KUKA KRL program: ps_geo_c1.src, ps_geo_c1.dat

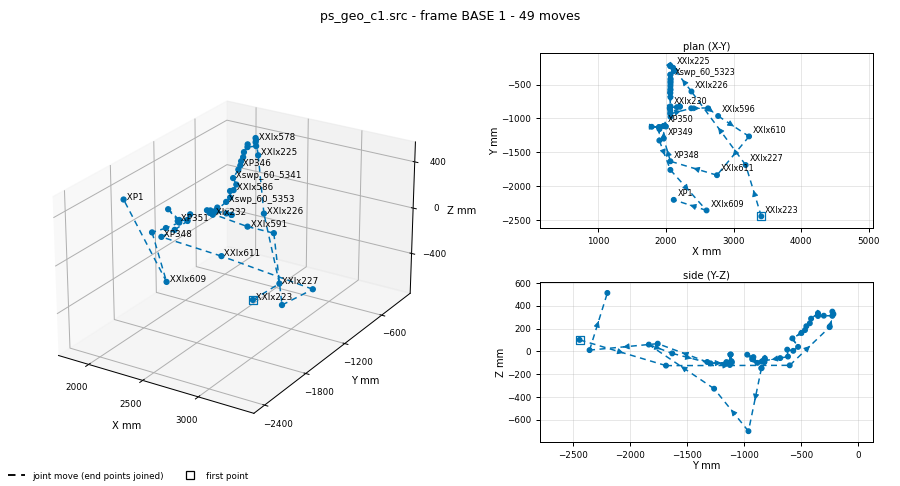
[picture p0: tool path of ps_geo_c1.src in frame BASE 1, 49 of 49 moves have a stored position in this frame; points joined in program order, loops and branches not executed]
--- ps_geo_c1.src ---
&ACCESS RVO1
&REL 105
&COMMENT Solda GUN C1 geometria
&PARAM DISKPATH = KRC:\R1\Program
DEF ps_geo_c1( )
;FOLD INI
  ;FOLD BASISTECH INI
    GLOBAL INTERRUPT DECL 3 WHEN $STOPMESS==TRUE DO IR_STOPM ( )
    INTERRUPT ON 3
    BAS (#INITMOV,0 )
  ;ENDFOLD (BASISTECH INI)
;FOLD SPOTTECH INI
USERSPOT(#INIT)
;ENDFOLD (SPOTTECH INI)
;FOLD GRIPPERTECH INI
USER_GRP(0,DUMMY,DUMMY,GDEFAULT)
;ENDFOLD (GRIPPERTECH INI)
  ;FOLD USER INI
    ;Make your modifications here

  ;ENDFOLD (USER INI)
;ENDFOLD (INI)

; Caracterização dos meios de produção:
; Versão Atual:
; 08/06/2013 12:00 Name: P13.050-R1 CHANGES: Solda Geometria Actros
; Gun C1 (F2 6640 0018 984)

chk_w2_wechs_ok ( )              ; CHECK C1

if MaxStandMenge (1) then
 MaxStandmengeErreicht (1)
endif

IF (NOT(GHOST())) THEN
if Elektrodenwechsel (1) then
 e_fraes2 ()
endif
ENDIF

;FOLD PTP Xlx223 CONT Vel=100 % P_OLP2 Tool[2]:GUN C1 Base[1]:Actros;%{PE}%R 8.2.20,%MKUKATPBASIS,%CMOVE,%VPTP,%P 1:PTP, 2:Xlx223, 3:C_DIS, 5:100, 7:P_OLP2
$BWDSTART=FALSE
PDAT_ACT=PP_OLP2
FDAT_ACT=FXlx223
BAS(#PTP_PARAMS,100)
PTP XXlx223 C_DIS
;ENDFOLD
;FOLD PTP Xlx227 CONT Vel=100 % P_OLP3 Tool[2]:GUN C1 Base[1]:Actros;%{PE}%R 8.2.20,%MKUKATPBASIS,%CMOVE,%VPTP,%P 1:PTP, 2:Xlx227, 3:C_DIS, 5:100, 7:P_OLP3
$BWDSTART=FALSE
PDAT_ACT=PP_OLP3
FDAT_ACT=FXlx227
BAS(#PTP_PARAMS,100)
PTP XXlx227 C_DIS
;ENDFOLD

;FOLD OUT 3339 'R1 solicita lib soldar geometria' State=TRUE ;%{PE}%R 8.2.20,%MKUKATPBASIS,%COUT,%VOUTX,%P 2:3339, 3:R1 solicita lib soldar geometria, 5:TRUE, 6:
$OUT[3339]=TRUE
;ENDFOLD
;FOLD WAIT FOR ( IN 3339 'Aguarda lib. Soldar geometria' );%{PE}%R 8.2.20,%MKUKATPBASIS,%CEXT_WAIT_FOR,%VEXT_WAIT_FOR,%P 2:, 4:, 5:$IN, 6:3339, 7:Aguarda lib. Soldar geometria, 9:
WAIT FOR  ( $IN[3339] )
;ENDFOLD
;FOLD OUT 3339 'R1 solicita lib soldar geometria' State=FALSE ;%{PE}%R 8.2.20,%MKUKATPBASIS,%COUT,%VOUTX,%P 2:3339, 3:R1 solicita lib soldar geometria, 5:FALSE, 6:
$OUT[3339]=FALSE
;ENDFOLD
;FOLD OUT 3348 'Fora area GEOBOX' State=FALSE ;%{PE}%R 8.2.20,%MKUKATPBASIS,%COUT,%VOUTX,%P 2:3348, 3:Fora area GEOBOX, 5:FALSE, 6:
$OUT[3348]=FALSE
;ENDFOLD

;FOLD PTP Xlx226 Vel=100 % P_OLP4 Tool[2]:GUN C1 Base[1]:Actros;%{PE}%R 8.2.20,%MKUKATPBASIS,%CMOVE,%VPTP,%P 1:PTP, 2:Xlx226, 3:, 5:100, 7:P_OLP4
$BWDSTART=FALSE
PDAT_ACT=PP_OLP4
FDAT_ACT=FXlx226
BAS(#PTP_PARAMS,100)
PTP XXlx226
;ENDFOLD

;FOLD Collision.Monitoring_AREA_6_On ;%{PE}%MKUKATPUSER
COLLSTOP( 12, 1 ) ;not Interrupt-Controlled
;ENDFOLD

;FOLD PTP Xlx225 CONT Vel=100 % P_OLP5 Tool[2]:GUN C1 Base[1]:Actros;%{PE}%R 8.2.20,%MKUKATPBASIS,%CMOVE,%VPTP,%P 1:PTP, 2:Xlx225, 3:C_DIS, 5:100, 7:P_OLP5
$BWDSTART=FALSE
PDAT_ACT=PP_OLP5
FDAT_ACT=FXlx225
BAS(#PTP_PARAMS,100)
PTP XXlx225 C_DIS
;ENDFOLD
;FOLD PTP Xlx578 CONT Vel=100 % PDAT1 Tool[2]:GUN C1 Base[1]:Actros;%{PE}%R 8.2.20,%MKUKATPBASIS,%CMOVE,%VPTP,%P 1:PTP, 2:Xlx578, 3:C_DIS, 5:100, 7:PDAT1
$BWDSTART=FALSE
PDAT_ACT=PPDAT1
FDAT_ACT=FXlx578
BAS(#PTP_PARAMS,100)
PTP XXlx578 C_DIS
;ENDFOLD

;FOLD ; swp_60_5311;%{PE}%R 8.2.20,%MKUKATPBASIS,%CCOMMENT,%VNORMAL,%P 2:swp_60_5311
;ENDFOLD
;FOLD PTP swp_60_5311 P_OLP6 SPOT Gun=1 RETR CLS PgNo1=26 ACTIVE=1 Tool[2]:GUN C1 Base[1]:Actros;%{PE}%R 8.2.2,%MKUKATPSPOT,%CSPOT,%VPTP,%P 1:PTP, 2:swp_60_5311, 3:, 5:100, 7:P_OLP6, 10:1, 12:#FIRST, 14:#CLO, 16:26, 18:1, 20:1, 22:0, 24:1, 25:S_OLP1
$BWDSTART=FALSE
PDAT_ACT=PP_OLP6
FDAT_ACT=Fswp_60_5311
BAS(#PTP_PARAMS,PP_OLP6.VEL)
S_ACT.GUN=1
S_ACT.PAIR=SDEFAULT.PAIR
S_ACT.RETR=#CLO
S_ACT.CLO_TM=1
S_ACT.PGNO1=26
S_ACT.PGNO2=SDEFAULT.PGNO2
S_ACT.PRESS1=SDEFAULT.PRESS1
S_ACT.PRESS2=SDEFAULT.PRESS2
S_READY=FALSE
PTP Xswp_60_5311
USERSPOT(#SPOT, S_ACT)
WAIT FOR S_READY
;ENDFOLD

;FOLD PTP Xlx583 CONT Vel=100 % PDAT6 Tool[2]:GUN C1 Base[1]:Actros;%{PE}%R 8.2.19,%MKUKATPBASIS,%CMOVE,%VPTP,%P 1:PTP, 2:Xlx583, 3:C_DIS, 5:100, 7:PDAT6
$BWDSTART=FALSE
PDAT_ACT=PPDAT6
FDAT_ACT=FXlx583
BAS(#PTP_PARAMS,100)
PTP XXlx583 C_DIS
;ENDFOLD
;FOLD PTP P347 CONT Vel=100 % PDAT39 Tool[2]:GUN C1 Base[1]:Actros;%{PE}%R 8.2.20,%MKUKATPBASIS,%CMOVE,%VPTP,%P 1:PTP, 2:P347, 3:C_DIS, 5:100, 7:PDAT39
$BWDSTART=FALSE
PDAT_ACT=PPDAT39
FDAT_ACT=FP347
BAS(#PTP_PARAMS,100)
PTP XP347 C_DIS
;ENDFOLD
;FOLD PTP Xlx584 CONT Vel=100 % PDAT7 Tool[2]:GUN C1 Base[1]:Actros;%{PE}%R 8.2.19,%MKUKATPBASIS,%CMOVE,%VPTP,%P 1:PTP, 2:Xlx584, 3:C_DIS, 5:100, 7:PDAT7
$BWDSTART=FALSE
PDAT_ACT=PPDAT7
FDAT_ACT=FXlx584
BAS(#PTP_PARAMS,100)
PTP XXlx584 C_DIS
;ENDFOLD

;FOLD ; swp_60_5317;%{PE}%R 8.2.20,%MKUKATPBASIS,%CCOMMENT,%VNORMAL,%P 2:swp_60_5317
;ENDFOLD
;FOLD PTP swp_60_5317 P_OLP42 SPOT Gun=1 RETR CLS PgNo1=27 ACTIVE=1 Tool[2]:GUN C1 Base[1]:Actros;%{PE}%R 8.2.2,%MKUKATPSPOT,%CSPOT,%VPTP,%P 1:PTP, 2:swp_60_5317, 3:, 5:100, 7:P_OLP42, 10:1, 12:#FIRST, 14:#CLO, 16:27, 18:1, 20:1, 22:0, 24:1, 25:S_OLP2
$BWDSTART=FALSE
PDAT_ACT=PP_OLP42
FDAT_ACT=Fswp_60_5317
BAS(#PTP_PARAMS,PP_OLP42.VEL)
S_ACT.GUN=1
S_ACT.PAIR=SDEFAULT.PAIR
S_ACT.RETR=#CLO
S_ACT.CLO_TM=1
S_ACT.PGNO1=27
S_ACT.PGNO2=SDEFAULT.PGNO2
S_ACT.PRESS1=SDEFAULT.PRESS1
S_ACT.PRESS2=SDEFAULT.PRESS2
S_READY=FALSE
PTP Xswp_60_5317
USERSPOT(#SPOT, S_ACT)
WAIT FOR S_READY
;ENDFOLD

;FOLD ; swp_60_5323;%{PE}%R 8.2.20,%MKUKATPBASIS,%CCOMMENT,%VNORMAL,%P 2:swp_60_5323
;ENDFOLD
;FOLD PTP swp_60_5323 P_OLP8 SPOT Gun=1 RETR CLS PgNo1=28 ACTIVE=1 Tool[2]:GUN C1 Base[1]:Actros;%{PE}%R 8.2.2,%MKUKATPSPOT,%CSPOT,%VPTP,%P 1:PTP, 2:swp_60_5323, 3:, 5:100, 7:P_OLP8, 10:1, 12:#FIRST, 14:#CLO, 16:28, 18:1, 20:1, 22:0, 24:1, 25:S_OLP3
$BWDSTART=FALSE
PDAT_ACT=PP_OLP8
FDAT_ACT=Fswp_60_5323
BAS(#PTP_PARAMS,PP_OLP8.VEL)
S_ACT.GUN=1
S_ACT.PAIR=SDEFAULT.PAIR
S_ACT.RETR=#CLO
S_ACT.CLO_TM=1
S_ACT.PGNO1=28
S_ACT.PGNO2=SDEFAULT.PGNO2
S_ACT.PRESS1=SDEFAULT.PRESS1
S_ACT.PRESS2=SDEFAULT.PRESS2
S_READY=FALSE
PTP Xswp_60_5323
USERSPOT(#SPOT, S_ACT)
WAIT FOR S_READY
;ENDFOLD

;FOLD PTP P345 CONT Vel=100 % PDAT37 Tool[2]:GUN C1 Base[1]:Actros;%{PE}%R 8.2.20,%MKUKATPBASIS,%CMOVE,%VPTP,%P 1:PTP, 2:P345, 3:C_DIS, 5:100, 7:PDAT37
$BWDSTART=FALSE
PDAT_ACT=PPDAT37
FDAT_ACT=FP345
BAS(#PTP_PARAMS,100)
PTP XP345 C_DIS
;ENDFOLD

;FOLD ; swp_60_5329;%{PE}%R 8.2.20,%MKUKATPBASIS,%CCOMMENT,%VNORMAL,%P 2:swp_60_5329
;ENDFOLD
;FOLD PTP swp_60_5329 P_OLP9 SPOT Gun=1 RETR CLS PgNo1=29 ACTIVE=1 Tool[2]:GUN C1 Base[1]:Actros;%{PE}%R 8.2.2,%MKUKATPSPOT,%CSPOT,%VPTP,%P 1:PTP, 2:swp_60_5329, 3:, 5:100, 7:P_OLP9, 10:1, 12:#FIRST, 14:#CLO, 16:29, 18:1, 20:1, 22:0, 24:1, 25:S_OLP4
$BWDSTART=FALSE
PDAT_ACT=PP_OLP9
FDAT_ACT=Fswp_60_5329
BAS(#PTP_PARAMS,PP_OLP9.VEL)
S_ACT.GUN=1
S_ACT.PAIR=SDEFAULT.PAIR
S_ACT.RETR=#CLO
S_ACT.CLO_TM=1
S_ACT.PGNO1=29
S_ACT.PGNO2=SDEFAULT.PGNO2
S_ACT.PRESS1=SDEFAULT.PRESS1
S_ACT.PRESS2=SDEFAULT.PRESS2
S_READY=FALSE
PTP Xswp_60_5329
USERSPOT(#SPOT, S_ACT)
WAIT FOR S_READY
;ENDFOLD

;FOLD PTP P346 CONT Vel=100 % PDAT38 Tool[2]:GUN C1 Base[1]:Actros;%{PE}%R 8.2.20,%MKUKATPBASIS,%CMOVE,%VPTP,%P 1:PTP, 2:P346, 3:C_DIS, 5:100, 7:PDAT38
$BWDSTART=FALSE
PDAT_ACT=PPDAT38
FDAT_ACT=FP346
BAS(#PTP_PARAMS,100)
PTP XP346 C_DIS
;ENDFOLD

;FOLD ; swp_60_5335;%{PE}%R 8.2.20,%MKUKATPBASIS,%CCOMMENT,%VNORMAL,%P 2:swp_60_5335
;ENDFOLD
;FOLD PTP swp_60_5335 P_OLP10 SPOT Gun=1 RETR CLS PgNo1=30 ACTIVE=1 Tool[2]:GUN C1 Base[1]:Actros;%{PE}%R 8.2.2,%MKUKATPSPOT,%CSPOT,%VPTP,%P 1:PTP, 2:swp_60_5335, 3:, 5:100, 7:P_OLP10, 10:1, 12:#FIRST, 14:#CLO, 16:30, 18:1, 20:1, 22:0, 24:1, 25:S_OLP5
$BWDSTART=FALSE
PDAT_ACT=PP_OLP10
FDAT_ACT=Fswp_60_5335
BAS(#PTP_PARAMS,PP_OLP10.VEL)
S_ACT.GUN=1
S_ACT.PAIR=SDEFAULT.PAIR
S_ACT.RETR=#CLO
S_ACT.CLO_TM=1
S_ACT.PGNO1=30
S_ACT.PGNO2=SDEFAULT.PGNO2
S_ACT.PRESS1=SDEFAULT.PRESS1
S_ACT.PRESS2=SDEFAULT.PRESS2
S_READY=FALSE
PTP Xswp_60_5335
USERSPOT(#SPOT, S_ACT)
WAIT FOR S_READY
;ENDFOLD

;FOLD ; swp_60_5341;%{PE}%R 8.2.20,%MKUKATPBASIS,%CCOMMENT,%VNORMAL,%P 2:swp_60_5341
;ENDFOLD
;FOLD PTP swp_60_5341 P_OLP11 SPOT Gun=1 RETR CLS PgNo1=31 ACTIVE=1 Tool[2]:GUN C1 Base[1]:Actros;%{PE}%R 8.2.2,%MKUKATPSPOT,%CSPOT,%VPTP,%P 1:PTP, 2:swp_60_5341, 3:, 5:100, 7:P_OLP11, 10:1, 12:#FIRST, 14:#CLO, 16:31, 18:1, 20:1, 22:0, 24:1, 25:S_OLP6
$BWDSTART=FALSE
PDAT_ACT=PP_OLP11
FDAT_ACT=Fswp_60_5341
BAS(#PTP_PARAMS,PP_OLP11.VEL)
S_ACT.GUN=1
S_ACT.PAIR=SDEFAULT.PAIR
S_ACT.RETR=#CLO
S_ACT.CLO_TM=1
S_ACT.PGNO1=31
S_ACT.PGNO2=SDEFAULT.PGNO2
S_ACT.PRESS1=SDEFAULT.PRESS1
S_ACT.PRESS2=SDEFAULT.PRESS2
S_READY=FALSE
PTP Xswp_60_5341
USERSPOT(#SPOT, S_ACT)
WAIT FOR S_READY
;ENDFOLD

;FOLD PTP Xlx585 CONT Vel=100 % PDAT8 Tool[2]:GUN C1 Base[1]:Actros;%{PE}%R 8.2.19,%MKUKATPBASIS,%CMOVE,%VPTP,%P 1:PTP, 2:Xlx585, 3:C_DIS, 5:100, 7:PDAT8
$BWDSTART=FALSE
PDAT_ACT=PPDAT8
FDAT_ACT=FXlx585
BAS(#PTP_PARAMS,100)
PTP XXlx585 C_DIS
;ENDFOLD
;FOLD PTP Xlx586 CONT Vel=100 % PDAT9 Tool[2]:GUN C1 Base[1]:Actros;%{PE}%R 8.2.19,%MKUKATPBASIS,%CMOVE,%VPTP,%P 1:PTP, 2:Xlx586, 3:C_DIS, 5:100, 7:PDAT9
$BWDSTART=FALSE
PDAT_ACT=PPDAT9
FDAT_ACT=FXlx586
BAS(#PTP_PARAMS,100)
PTP XXlx586 C_DIS
;ENDFOLD

;FOLD ; swp_60_5347;%{PE}%R 8.2.20,%MKUKATPBASIS,%CCOMMENT,%VNORMAL,%P 2:swp_60_5347
;ENDFOLD
;FOLD PTP swp_60_5347 P_OLP12 SPOT Gun=1 RETR CLS PgNo1=32 ACTIVE=1 Tool[2]:GUN C1 Base[1]:Actros;%{PE}%R 8.2.2,%MKUKATPSPOT,%CSPOT,%VPTP,%P 1:PTP, 2:swp_60_5347, 3:, 5:100, 7:P_OLP12, 10:1, 12:#FIRST, 14:#CLO, 16:32, 18:1, 20:1, 22:0, 24:1, 25:S_OLP7
$BWDSTART=FALSE
PDAT_ACT=PP_OLP12
FDAT_ACT=Fswp_60_5347
BAS(#PTP_PARAMS,PP_OLP12.VEL)
S_ACT.GUN=1
S_ACT.PAIR=SDEFAULT.PAIR
S_ACT.RETR=#CLO
S_ACT.CLO_TM=1
S_ACT.PGNO1=32
S_ACT.PGNO2=SDEFAULT.PGNO2
S_ACT.PRESS1=SDEFAULT.PRESS1
S_ACT.PRESS2=SDEFAULT.PRESS2
S_READY=FALSE
PTP Xswp_60_5347
USERSPOT(#SPOT, S_ACT)
WAIT FOR S_READY
;ENDFOLD

;FOLD PTP Xlx587 CONT Vel=100 % PDAT10 Tool[2]:GUN C1 Base[1]:Actros;%{PE}%R 8.2.19,%MKUKATPBASIS,%CMOVE,%VPTP,%P 1:PTP, 2:Xlx587, 3:C_DIS, 5:100, 7:PDAT10
$BWDSTART=FALSE
PDAT_ACT=PPDAT10
FDAT_ACT=FXlx587
BAS(#PTP_PARAMS,100)
PTP XXlx587 C_DIS
;ENDFOLD

;FOLD ; swp_60_5353;%{PE}%R 8.2.20,%MKUKATPBASIS,%CCOMMENT,%VNORMAL,%P 2:swp_60_5353
;ENDFOLD
;FOLD PTP swp_60_5353 P_OLP13 SPOT Gun=1 RETR CLS PgNo1=33 ACTIVE=1 Tool[2]:GUN C1 Base[1]:Actros;%{PE}%R 8.2.2,%MKUKATPSPOT,%CSPOT,%VPTP,%P 1:PTP, 2:swp_60_5353, 3:, 5:100, 7:P_OLP13, 10:1, 12:#FIRST, 14:#CLO, 16:33, 18:1, 20:1, 22:0, 24:1, 25:S_OLP8
$BWDSTART=FALSE
PDAT_ACT=PP_OLP13
FDAT_ACT=Fswp_60_5353
BAS(#PTP_PARAMS,PP_OLP13.VEL)
S_ACT.GUN=1
S_ACT.PAIR=SDEFAULT.PAIR
S_ACT.RETR=#CLO
S_ACT.CLO_TM=1
S_ACT.PGNO1=33
S_ACT.PGNO2=SDEFAULT.PGNO2
S_ACT.PRESS1=SDEFAULT.PRESS1
S_ACT.PRESS2=SDEFAULT.PRESS2
S_READY=FALSE
PTP Xswp_60_5353
USERSPOT(#SPOT, S_ACT)
WAIT FOR S_READY
;ENDFOLD

;FOLD PTP Xlx230 CONT Vel=100 % P_OLP14 Tool[2]:GUN C1 Base[1]:Actros;%{PE}%R 8.2.19,%MKUKATPBASIS,%CMOVE,%VPTP,%P 1:PTP, 2:Xlx230, 3:C_DIS, 5:100, 7:P_OLP14
$BWDSTART=FALSE
PDAT_ACT=PP_OLP14
FDAT_ACT=FXlx230
BAS(#PTP_PARAMS,100)
PTP XXlx230 C_DIS
;ENDFOLD

;FOLD PTP Xlx231 CONT Vel=100 % P_OLP43 Tool[2]:GUN C1 Base[1]:Actros;%{PE}%R 8.2.20,%MKUKATPBASIS,%CMOVE,%VPTP,%P 1:PTP, 2:Xlx231, 3:C_DIS, 5:100, 7:P_OLP43
$BWDSTART=FALSE
PDAT_ACT=PP_OLP43
FDAT_ACT=FXlx231
BAS(#PTP_PARAMS,100)
PTP XXlx231 C_DIS
;ENDFOLD
;FOLD PTP Xlx232 CONT Vel=100 % P_OLP44 Tool[2]:GUN C1 Base[1]:Actros;%{PE}%R 8.2.20,%MKUKATPBASIS,%CMOVE,%VPTP,%P 1:PTP, 2:Xlx232, 3:C_DIS, 5:100, 7:P_OLP44
$BWDSTART=FALSE
PDAT_ACT=PP_OLP44
FDAT_ACT=FXlx232
BAS(#PTP_PARAMS,100)
PTP XXlx232 C_DIS
;ENDFOLD
;FOLD Collision.Monitoring_AREA_6_Off . ;%{PE}%MKUKATPUSER
COLLSTOP( 12, 2+0 )
;ENDFOLD

;FOLD PTP Xlx229 CONT Vel=100 % P_OLP16 Tool[2]:GUN C1 Base[1]:Actros;%{PE}%R 8.2.19,%MKUKATPBASIS,%CMOVE,%VPTP,%P 1:PTP, 2:Xlx229, 3:C_DIS, 5:100, 7:P_OLP16
$BWDSTART=FALSE
PDAT_ACT=PP_OLP16
FDAT_ACT=FXlx229
BAS(#PTP_PARAMS,100)
PTP XXlx229 C_DIS
;ENDFOLD
;FOLD PTP Xlx228 CONT Vel=100 % P_OLP17 Tool[2]:GUN C1 Base[1]:Actros;%{PE}%R 8.2.19,%MKUKATPBASIS,%CMOVE,%VPTP,%P 1:PTP, 2:Xlx228, 3:C_DIS, 5:100, 7:P_OLP17
$BWDSTART=FALSE
PDAT_ACT=PP_OLP17
FDAT_ACT=FXlx228
BAS(#PTP_PARAMS,100)
PTP XXlx228 C_DIS
;ENDFOLD

;FOLD ; swp_60_5359;%{PE}%R 8.2.20,%MKUKATPBASIS,%CCOMMENT,%VNORMAL,%P 2:swp_60_5359
;ENDFOLD
;FOLD PTP swp_60_5359 P_OLP18 SPOT Gun=1 RETR CLS PgNo1=34 ACTIVE=1 Tool[2]:GUN C1 Base[1]:Actros;%{PE}%R 8.2.2,%MKUKATPSPOT,%CSPOT,%VPTP,%P 1:PTP, 2:swp_60_5359, 3:, 5:100, 7:P_OLP18, 10:1, 12:#FIRST, 14:#CLO, 16:34, 18:1, 20:1, 22:0, 24:1, 25:S_OLP9
$BWDSTART=FALSE
PDAT_ACT=PP_OLP18
FDAT_ACT=Fswp_60_5359
BAS(#PTP_PARAMS,PP_OLP18.VEL)
S_ACT.GUN=1
S_ACT.PAIR=SDEFAULT.PAIR
S_ACT.RETR=#CLO
S_ACT.CLO_TM=1
S_ACT.PGNO1=34
S_ACT.PGNO2=SDEFAULT.PGNO2
S_ACT.PRESS1=SDEFAULT.PRESS1
S_ACT.PRESS2=SDEFAULT.PRESS2
S_READY=FALSE
PTP Xswp_60_5359
USERSPOT(#SPOT, S_ACT)
WAIT FOR S_READY
;ENDFOLD

;FOLD PTP Xlx232 CONT Vel=100 % P_OLP19 Tool[2]:GUN C1 Base[1]:Actros;%{PE}%R8.2,%MKUKATPBASIS,%CMOVE,%VPTP,%P 1:PTP, 2:Xlx232, 3:C_DIS, 5:100, 7:P_OLP19
$BWDSTART = FALSE
PDAT_ACT= PP_OLP19
FDAT_ACT= Flx232
BAS(#PTP_PARAMS,100)
PTP Xlx232 C_DIS
;ENDFOLD
;FOLD PTP Xlx595 CONT Vel=100 % PDAT18 Tool[2]:GUN C1 Base[1]:Actros;%{PE}%R 8.2.19,%MKUKATPBASIS,%CMOVE,%VPTP,%P 1:PTP, 2:Xlx595, 3:C_DIS, 5:100, 7:PDAT18
$BWDSTART=FALSE
PDAT_ACT=PPDAT18
FDAT_ACT=FXlx595
BAS(#PTP_PARAMS,100)
PTP XXlx595 C_DIS
;ENDFOLD

;FOLD ; swp_60_5367;%{PE}%R 8.2.20,%MKUKATPBASIS,%CCOMMENT,%VNORMAL,%P 2:swp_60_5367
;ENDFOLD
;FOLD PTP swp_60_5367 P_OLP41 SPOT Gun=1 RETR CLS PgNo1=35 ACTIVE=1 Tool[2]:GUN C1 Base[1]:Actros;%{PE}%R 8.2.2,%MKUKATPSPOT,%CSPOT,%VPTP,%P 1:PTP, 2:swp_60_5367, 3:, 5:100, 7:P_OLP41, 10:1, 12:#FIRST, 14:#CLO, 16:35, 18:1, 20:1, 22:0, 24:1, 25:S_OLP14
$BWDSTART=FALSE
PDAT_ACT=PP_OLP41
FDAT_ACT=Fswp_60_5367
BAS(#PTP_PARAMS,PP_OLP41.VEL)
S_ACT.GUN=1
S_ACT.PAIR=SDEFAULT.PAIR
S_ACT.RETR=#CLO
S_ACT.CLO_TM=1
S_ACT.PGNO1=35
S_ACT.PGNO2=SDEFAULT.PGNO2
S_ACT.PRESS1=SDEFAULT.PRESS1
S_ACT.PRESS2=SDEFAULT.PRESS2
S_READY=FALSE
PTP Xswp_60_5367
USERSPOT(#SPOT, S_ACT)
WAIT FOR S_READY
;ENDFOLD

;FOLD PTP Xlx592 CONT Vel=100 % PDAT15 Tool[2]:GUN C1 Base[1]:Actros;%{PE}%R 8.2.19,%MKUKATPBASIS,%CMOVE,%VPTP,%P 1:PTP, 2:Xlx592, 3:C_DIS, 5:100, 7:PDAT15
$BWDSTART=FALSE
PDAT_ACT=PPDAT15
FDAT_ACT=FXlx592
BAS(#PTP_PARAMS,100)
PTP XXlx592 C_DIS
;ENDFOLD
;FOLD PTP Xlx591 CONT Vel=100 % PDAT14 Tool[2]:GUN C1 Base[1]:Actros;%{PE}%R 8.2.19,%MKUKATPBASIS,%CMOVE,%VPTP,%P 1:PTP, 2:Xlx591, 3:C_DIS, 5:100, 7:PDAT14
$BWDSTART=FALSE
PDAT_ACT=PPDAT14
FDAT_ACT=FXlx591
BAS(#PTP_PARAMS,100)
PTP XXlx591 C_DIS
;ENDFOLD
;FOLD PTP Xlx594 CONT Vel=100 % PDAT17 Tool[2]:GUN C1 Base[1]:Actros;%{PE}%R 8.2.19,%MKUKATPBASIS,%CMOVE,%VPTP,%P 1:PTP, 2:Xlx594, 3:C_DIS, 5:100, 7:PDAT17
$BWDSTART=FALSE
PDAT_ACT=PPDAT17
FDAT_ACT=FXlx594
BAS(#PTP_PARAMS,100)
PTP XXlx594 C_DIS
;ENDFOLD
;FOLD PTP Xlx596 CONT Vel=100 % PDAT19 Tool[2]:GUN C1 Base[1]:Actros;%{PE}%R 8.2.19,%MKUKATPBASIS,%CMOVE,%VPTP,%P 1:PTP, 2:Xlx596, 3:C_DIS, 5:100, 7:PDAT19
$BWDSTART=FALSE
PDAT_ACT=PPDAT19
FDAT_ACT=FXlx596
BAS(#PTP_PARAMS,100)
PTP XXlx596 C_DIS
;ENDFOLD
;FOLD PTP Xlx610 CONT Vel=100 % PDAT33 Tool[2]:GUN C1 Base[1]:Actros;%{PE}%R 8.2.19,%MKUKATPBASIS,%CMOVE,%VPTP,%P 1:PTP, 2:Xlx610, 3:C_DIS, 5:100, 7:PDAT33
$BWDSTART=FALSE
PDAT_ACT=PPDAT33
FDAT_ACT=FXlx610
BAS(#PTP_PARAMS,100)
PTP XXlx610 C_DIS
;ENDFOLD
;FOLD PTP Xlx611 CONT Vel=100 % PDAT34 Tool[2]:GUN C1 Base[1]:Actros;%{PE}%R 8.2.19,%MKUKATPBASIS,%CMOVE,%VPTP,%P 1:PTP, 2:Xlx611, 3:C_DIS, 5:100, 7:PDAT34
$BWDSTART=FALSE
PDAT_ACT=PPDAT34
FDAT_ACT=FXlx611
BAS(#PTP_PARAMS,100)
PTP XXlx611 C_DIS
;ENDFOLD
;FOLD PTP P348 CONT Vel=100 % PDAT40 Tool[2]:GUN C1 Base[1]:Actros;%{PE}%R 8.2.20,%MKUKATPBASIS,%CMOVE,%VPTP,%P 1:PTP, 2:P348, 3:C_DIS, 5:100, 7:PDAT40
$BWDSTART=FALSE
PDAT_ACT=PPDAT40
FDAT_ACT=FP348
BAS(#PTP_PARAMS,100)
PTP XP348 C_DIS
;ENDFOLD
;FOLD PTP P349 CONT Vel=100 % PDAT41 Tool[2]:GUN C1 Base[1]:Actros;%{PE}%R 8.2.20,%MKUKATPBASIS,%CMOVE,%VPTP,%P 1:PTP, 2:P349, 3:C_DIS, 5:100, 7:PDAT41
$BWDSTART=FALSE
PDAT_ACT=PPDAT41
FDAT_ACT=FP349
BAS(#PTP_PARAMS,100)
PTP XP349 C_DIS
;ENDFOLD
;FOLD PTP P350 PDAT42 RETR CLS Gun=1 Tool[2]:GUN C1 Base[1]:Actros;%{PE}%R 8.2.2,%MKUKATPSPOT,%CRETR,%VPTP,%P 1:PTP, 2:P350, 3:, 5:100, 7:PDAT42, 9:#CLO, 11:1, 13:#FIRST
$BWDSTART=FALSE
PDAT_ACT=PPDAT42
FDAT_ACT=FP350
BAS(#PTP_PARAMS,PPDAT42.VEL)
S_ACT.GUN=1
S_ACT.PAIR=#FIRST
S_ACT.RETR=#CLO
S_READY=FALSE
PTP XP350
USERSPOT(#RETR, S_ACT)
WAIT FOR S_READY
;ENDFOLD

;FOLD ; swp_60_5377;%{PE}%R 8.2.20,%MKUKATPBASIS,%CCOMMENT,%VNORMAL,%P 2:swp_60_5377
;ENDFOLD
;FOLD PTP SWP_60_5377 PDAT43 SPOT Gun=1 RETR CLS PgNo1=36 ACTIVE=1 Tool[2]:GUN C1 Base[1]:Actros;%{PE}%R 8.2.2,%MKUKATPSPOT,%CSPOT,%VPTP,%P 1:PTP, 2:SWP_60_5377, 3:, 5:100, 7:PDAT43, 10:1, 12:#FIRST, 14:#CLO, 16:36, 18:1, 20:0, 22:0, 24:1, 25:SDAT1
$BWDSTART=FALSE
PDAT_ACT=PPDAT43
FDAT_ACT=FSWP_60_5377
BAS(#PTP_PARAMS,PPDAT43.VEL)
S_ACT.GUN=1
S_ACT.PAIR=SDEFAULT.PAIR
S_ACT.RETR=#CLO
S_ACT.CLO_TM=1
S_ACT.PGNO1=36
S_ACT.PGNO2=SDEFAULT.PGNO2
S_ACT.PRESS1=SDEFAULT.PRESS1
S_ACT.PRESS2=SDEFAULT.PRESS2
S_READY=FALSE
PTP XSWP_60_5377
USERSPOT(#SPOT, S_ACT)
WAIT FOR S_READY
;ENDFOLD

;FOLD PTP P456 CONT Vel=100 % PDAT44 Tool[2]:GUN C1 Base[1]:Actros;%{PE}%R 8.2.20,%MKUKATPBASIS,%CMOVE,%VPTP,%P 1:PTP, 2:P456, 3:C_DIS, 5:100, 7:PDAT44
$BWDSTART=FALSE
PDAT_ACT=PPDAT44
FDAT_ACT=FP456
BAS(#PTP_PARAMS,100)
PTP XP456 C_DIS
;ENDFOLD
;FOLD PTP P351 CONT Vel=100 % PDAT45 Tool[2]:GUN C1 Base[1]:Actros;%{PE}%R 8.2.20,%MKUKATPBASIS,%CMOVE,%VPTP,%P 1:PTP, 2:P351, 3:C_DIS, 5:100, 7:PDAT45
$BWDSTART=FALSE
PDAT_ACT=PPDAT45
FDAT_ACT=FP351
BAS(#PTP_PARAMS,100)
PTP XP351 C_DIS
;ENDFOLD
;FOLD PTP P352 CONT Vel=100 % PDAT46 Tool[2]:GUN C1 Base[1]:Actros;%{PE}%R 8.2.20,%MKUKATPBASIS,%CMOVE,%VPTP,%P 1:PTP, 2:P352, 3:C_DIS, 5:100, 7:PDAT46
$BWDSTART=FALSE
PDAT_ACT=PPDAT46
FDAT_ACT=FP352
BAS(#PTP_PARAMS,100)
PTP XP352 C_DIS
;ENDFOLD

;FOLD ; swp_60_5387;%{PE}%R 8.2.20,%MKUKATPBASIS,%CCOMMENT,%VNORMAL,%P 2:swp_60_5387
;ENDFOLD
;FOLD PTP SWP_60_5387 PDAT47 SPOT Gun=1 RETR CLS PgNo1=37 ACTIVE=1 Tool[2]:GUN C1 Base[1]:Actros;%{PE}%R 8.2.2,%MKUKATPSPOT,%CSPOT,%VPTP,%P 1:PTP, 2:SWP_60_5387, 3:, 5:100, 7:PDAT47, 10:1, 12:#FIRST, 14:#CLO, 16:37, 18:1, 20:0, 22:0, 24:1, 25:SDAT2
$BWDSTART=FALSE
PDAT_ACT=PPDAT47
FDAT_ACT=FSWP_60_5387
BAS(#PTP_PARAMS,PPDAT47.VEL)
S_ACT.GUN=1
S_ACT.PAIR=SDEFAULT.PAIR
S_ACT.RETR=#CLO
S_ACT.CLO_TM=1
S_ACT.PGNO1=37
S_ACT.PGNO2=SDEFAULT.PGNO2
S_ACT.PRESS1=SDEFAULT.PRESS1
S_ACT.PRESS2=SDEFAULT.PRESS2
S_READY=FALSE
PTP XSWP_60_5387
USERSPOT(#SPOT, S_ACT)
WAIT FOR S_READY
;ENDFOLD

;FOLD PTP P455 CONT Vel=100 % PDAT48 Tool[2]:GUN C1 Base[1]:Actros;%{PE}%R 8.2.20,%MKUKATPBASIS,%CMOVE,%VPTP,%P 1:PTP, 2:P455, 3:C_DIS, 5:100, 7:PDAT48
$BWDSTART=FALSE
PDAT_ACT=PPDAT48
FDAT_ACT=FP455
BAS(#PTP_PARAMS,100)
PTP XP455 C_DIS
;ENDFOLD
;FOLD PTP P457 CONT Vel=100 % PDAT49 Tool[2]:GUN C1 Base[1]:Actros;%{PE}%R 8.2.20,%MKUKATPBASIS,%CMOVE,%VPTP,%P 1:PTP, 2:P457, 3:C_DIS, 5:100, 7:PDAT49
$BWDSTART=FALSE
PDAT_ACT=PPDAT49
FDAT_ACT=FP457
BAS(#PTP_PARAMS,100)
PTP XP457 C_DIS
;ENDFOLD
;FOLD PTP P458 CONT Vel=100 % PDAT50 Tool[2]:GUN C1 Base[1]:Actros;%{PE}%R 8.2.20,%MKUKATPBASIS,%CMOVE,%VPTP,%P 1:PTP, 2:P458, 3:C_DIS, 5:100, 7:PDAT50
$BWDSTART=FALSE
PDAT_ACT=PPDAT50
FDAT_ACT=FP458
BAS(#PTP_PARAMS,100)
PTP XP458 C_DIS
;ENDFOLD
;FOLD PTP Xlx609 CONT Vel=100 % PDAT32 Tool[2]:GUN C1 Base[1]:Actros;%{PE}%R 8.2.20,%MKUKATPBASIS,%CMOVE,%VPTP,%P 1:PTP, 2:Xlx609, 3:C_DIS, 5:100, 7:PDAT32
$BWDSTART=FALSE
PDAT_ACT=PPDAT32
FDAT_ACT=FXlx609
BAS(#PTP_PARAMS,100)
PTP XXlx609 C_DIS
;ENDFOLD
;FOLD PTP P1 Vel=100 % PDAT53 Tool[2]:GUN C1 Base[1]:Actros;%{PE}%R 8.2.20,%MKUKATPBASIS,%CMOVE,%VPTP,%P 1:PTP, 2:P1, 3:, 5:100, 7:PDAT53
$BWDSTART=FALSE
PDAT_ACT=PPDAT53
FDAT_ACT=FP1
BAS(#PTP_PARAMS,100)
PTP XP1
;ENDFOLD

;FOLD OUT 3348 'Fora area GEOBOX' State=TRUE ;%{PE}%R 8.2.20,%MKUKATPBASIS,%COUT,%VOUTX,%P 2:3348, 3:Fora area GEOBOX, 5:TRUE, 6:
$OUT[3348]=TRUE
;ENDFOLD

IF (NOT(GHOST())) THEN
if FraesAnf (1) then
 f_fraes2 ()
endif
ENDIF
END

--- ps_geo_c1.dat ---
&ACCESS RVO1
&REL 105
&COMMENT Solda GUN C1 geometria
&PARAM DISKPATH = KRC:\R1\Program
DEFDAT  ps_geo_c1
;FOLD EXTERNAL DECLARATIONS;%{PE}%MKUKATPBASIS,%CEXT,%VCOMMON,%P
;FOLD GRIPPERTECH EXT
EXT  H50 (INT  :IN,INT  :IN,INT  :IN,GRP_TYP  :IN )
;ENDFOLD (GRIPPERTECH EXT)
;FOLD SPOTTECH EXT
EXT  USERSPOT (S_COMMAND  :IN,SPOT_TYPE  :IN )
;ENDFOLD (SPOTTECH EXT)
;FOLD BASISTECH EXT;%{PE}%MKUKATPBASIS,%CEXT,%VEXT,%P
EXT  BAS (BAS_COMMAND  :IN,REAL  :IN )
DECL INT SUCCESS
;ENDFOLD (BASISTECH EXT)
;FOLD USER EXT;%{E}%MKUKATPUSER,%CEXT,%VEXT,%P
;Make your modifications here

;ENDFOLD (USER EXT)
;ENDFOLD (EXTERNAL DECLARATIONS)

;# ============ START PATH : swp_p13050r1_l_geo_c1 =============
DECL PDAT PP_OLP2={VEL 100.0,ACC 100.0,APO_DIST 100.0,APO_MODE #CDIS}
DECL PDAT PP_OLP3={VEL 100.0,ACC 100.0,APO_DIST 100.0,APO_MODE #CDIS}
DECL PDAT PP_OLP4={VEL 100.0,ACC 100.0,APO_DIST 100.0,APO_MODE #CDIS}
DECL PDAT PP_OLP5={VEL 100.0,ACC 100.0,APO_DIST 100.0,APO_MODE #CDIS}
DECL FDAT Fswp_60_5311={TOOL_NO 2,BASE_NO 1,IPO_FRAME #BASE,POINT2[] " ",TQ_STATE FALSE}
DECL PDAT PP_OLP6={VEL 100.0,ACC 100.0,APO_DIST 0.0}
DECL SPOT_TYPE SS_OLP1={GUN 1,PAIR #FIRST,RETR #CLO,CLO_TM 0,PGNO1 1,PRESS1 1.0,PGNO2 0,PRESS2 0.0}
DECL E6POS Xswp_60_5311={X 2065.98511,Y -226.899902,Z 349.511993,A 110.327499,B -85.6865234,C 69.4538727,S 2,T 42,E1 -4474.354,E2 0.0,E3 0.0,E4 0.0,E5 0.0,E6 0.0}
DECL FDAT Fswp_60_5317={TOOL_NO 2,BASE_NO 1,IPO_FRAME #BASE,POINT2[] " ",TQ_STATE FALSE}
DECL SPOT_TYPE SS_OLP2={GUN 1,PAIR #FIRST,RETR #CLO,CLO_TM 0,PGNO1 1,PRESS1 1.0,PGNO2 0,PRESS2 0.0}
DECL E6POS Xswp_60_5317={X 2067.58789,Y -353.265594,Z 335.725708,A -98.2681732,B -88.2489166,C -79.6126328,S 2,T 42,E1 -4219.60889,E2 0.0,E3 0.0,E4 0.0,E5 0.0,E6 0.0}
DECL FDAT Fswp_60_5323={TOOL_NO 2,BASE_NO 1,IPO_FRAME #BASE,POINT2[] " ",TQ_STATE FALSE}
DECL PDAT PP_OLP8={VEL 100.0,ACC 100.0,APO_DIST 0.0}
DECL SPOT_TYPE SS_OLP3={GUN 1,PAIR #FIRST,RETR #CLO,CLO_TM 0,PGNO1 1,PRESS1 1.0,PGNO2 0,PRESS2 0.0}
DECL E6POS Xswp_60_5323={X 2069.21704,Y -413.284393,Z 287.633209,A -84.5369034,B -66.7329865,C -93.644577,S 2,T 42,E1 -4219.93799,E2 0.0,E3 0.0,E4 0.0,E5 0.0,E6 0.0}
DECL FDAT Fswp_60_5329={TOOL_NO 2,BASE_NO 1,IPO_FRAME #BASE,POINT2[] " ",TQ_STATE FALSE}
DECL PDAT PP_OLP9={VEL 100.0,ACC 100.0,APO_DIST 0.0}
DECL SPOT_TYPE SS_OLP4={GUN 1,PAIR #FIRST,RETR #CLO,CLO_TM 0,PGNO1 1,PRESS1 1.0,PGNO2 0,PRESS2 0.0}
DECL E6POS Xswp_60_5329={X 2068.11792,Y -455.172089,Z 221.144104,A -83.784668,B -70.5104675,C -94.3365021,S 2,T 42,E1 -4219.93799,E2 0.0,E3 0.0,E4 0.0,E5 0.0,E6 0.0}
DECL FDAT Fswp_60_5335={TOOL_NO 2,BASE_NO 1,IPO_FRAME #BASE,POINT2[] " ",TQ_STATE FALSE}
DECL PDAT PP_OLP10={VEL 100.0,ACC 100.0,APO_DIST 0.0}
DECL SPOT_TYPE SS_OLP5={GUN 1,PAIR #FIRST,RETR #CLO,CLO_TM 0,PGNO1 1,PRESS1 1.0,PGNO2 0,PRESS2 0.0}
DECL E6POS Xswp_60_5335={X 2068.32104,Y -498.486511,Z 162.031601,A -83.1203003,B -73.1582031,C -94.9776001,S 2,T 42,E1 -4219.93799,E2 0.0,E3 0.0,E4 0.0,E5 0.0,E6 0.0}
DECL FDAT Fswp_60_5341={TOOL_NO 2,BASE_NO 1,IPO_FRAME #BASE,POINT2[] " "}
DECL PDAT PP_OLP11={VEL 100.0,ACC 100.0,APO_DIST 0.0}
DECL SPOT_TYPE SS_OLP6={GUN 1,PAIR #FIRST,RETR #CLO,CLO_TM 0,PGNO1 1,PRESS1 1.0,PGNO2 0,PRESS2 0.0}
DECL E6POS Xswp_60_5341={X 2067.21704,Y -577.190186,Z 114.618599,A -85.77388,B -55.6890182,C -92.5561829,S 2,T 10,E1 -4219.93799,E2 0.0,E3 0.0,E4 0.0,E5 0.0,E6 0.0}
DECL FDAT Fswp_60_5347={TOOL_NO 2,BASE_NO 1,IPO_FRAME #BASE,POINT2[] " ",TQ_STATE FALSE}
DECL PDAT PP_OLP12={VEL 100.0,ACC 100.0,APO_DIST 0.0}
DECL SPOT_TYPE SS_OLP7={GUN 1,PAIR #FIRST,RETR #CLO,CLO_TM 0,PGNO1 1,PRESS1 1.0,PGNO2 0,PRESS2 0.0}
DECL E6POS Xswp_60_5347={X 2066.55298,Y -622.881287,Z 15.8281803,A -85.6193771,B -57.4586182,C -92.6872101,S 2,T 10,E1 -4219.9458,E2 0.0,E3 0.0,E4 0.0,E5 0.0,E6 0.0}
DECL FDAT Fswp_60_5353={TOOL_NO 2,BASE_NO 1,IPO_FRAME #BASE,POINT2[] " "}
DECL PDAT PP_OLP13={VEL 100.0,ACC 100.0,APO_DIST 0.0}
DECL SPOT_TYPE SS_OLP8={GUN 1,PAIR #FIRST,RETR #CLO,CLO_TM 0,PGNO1 1,PRESS1 1.0,PGNO2 0,PRESS2 0.0}
DECL E6POS Xswp_60_5353={X 2067.23193,Y -684.528625,Z -58.5064888,A -86.9186478,B -33.8480606,C -91.7377472,S 2,T 10,E1 -4219.99512,E2 0.0,E3 0.0,E4 0.0,E5 0.0,E6 0.0}
DECL PDAT PP_OLP14={VEL 100.0,ACC 100.0,APO_DIST 100.0,APO_MODE #CDIS}
DECL PDAT PP_OLP16={VEL 100.0,ACC 100.0,APO_DIST 100.0,APO_MODE #CDIS}
DECL PDAT PP_OLP17={VEL 100.0,ACC 100.0,APO_DIST 100.0,APO_MODE #CDIS}
DECL FDAT Fswp_60_5359={TOOL_NO 2,BASE_NO 1,IPO_FRAME #BASE,POINT2[] " ",TQ_STATE FALSE}
DECL PDAT PP_OLP18={VEL 100.0,ACC 100.0,APO_DIST 0.0}
DECL SPOT_TYPE SS_OLP9={GUN 1,PAIR #FIRST,RETR #CLO,CLO_TM 0,PGNO1 1,PRESS1 1.0,PGNO2 0,PRESS2 0.0}
DECL E6POS Xswp_60_5359={X 2067.65308,Y -819.673706,Z -59.9566994,A 89.9988708,B -35.2867393,C 90.0017166,S 2,T 42,E1 -4487.30518,E2 0.0,E3 0.0,E4 0.0,E5 0.0,E6 0.0}
DECL FDAT Flx232={TOOL_NO 2,BASE_NO 1,IPO_FRAME #BASE,POINT2[] " "}
DECL PDAT PP_OLP19={VEL 100.0,ACC 100.0,APO_DIST 100.0,APO_MODE #CDIS}
DECL E6POS Xlx232={X 2065.2561,Y -885.252014,Z -100.142998,A 90.0,B -35.6880989,C 90.0,S 2,T 42,E1 -4487.2998,E2 0.0,E3 0.0,E4 0.0,E5 0.0,E6 0.0}
DECL FDAT Fswp_60_5367={TOOL_NO 2,BASE_NO 1,IPO_FRAME #BASE,POINT2[] " "}
DECL SPOT_TYPE SS_OLP10={GUN 1,PAIR #FIRST,RETR #CLO,CLO_TM 0,PGNO1 1,PRESS1 1.0,PGNO2 0,PRESS2 0.0}
DECL E6POS Xswp_60_5367={X 2067.479,Y -973.934082,Z -28.4924908,A 89.9911804,B -81.1077728,C 90.0090179,S 2,T 42,E1 -4487.2998,E2 0.0,E3 0.0,E4 0.0,E5 0.0,E6 0.0}
DECL FDAT Fswp_60_5377={TOOL_NO 2,BASE_NO 1,IPO_FRAME #BASE,POINT2[] " "}
DECL SPOT_TYPE SS_OLP11={GUN 1,PAIR #FIRST,RETR #CLO,CLO_TM 0,PGNO1 1,PRESS1 1.0,PGNO2 0,PRESS2 0.0}
DECL E6POS Xswp_60_5377={X 2000.44202,Y -1118.71997,Z -26.2877502,A -0.164200798,B -46.8474388,C 88.6065521,S 2,T 2,E1 -3882.23608,E2 0.0,E3 0.0,E4 0.0,E5 0.0,E6 0.0}
DECL SPOT_TYPE SS_OLP12={GUN 1,PAIR #FIRST,RETR #CLO,CLO_TM 0,PGNO1 1,PRESS1 1.0,PGNO2 0,PRESS2 0.0}
DECL BASIS_SUGG_T LAST_BASIS={POINT1[] "P0                      ",POINT2[] "P0                      ",CP_PARAMS[] "CPDAT0                  ",PTP_PARAMS[] "PDAT0                   ",CONT[] "                        ",CP_VEL[] "2.0                     ",PTP_VEL[] " 100                    ",SYNC_PARAMS[] "SYNCDAT                 ",SPL_NAME[] "S0                      "}
DECL E6POS XXLX223={X 3409.55396,Y -2445.41089,Z 101.454399,A 10.5907497,B 25.0754108,C 8.57579041,S 2,T 2,E1 -2854.21997,E2 0.0,E3 0.0,E4 0.0,E5 0.0,E6 0.0}
DECL FDAT FXlx223={TOOL_NO 2,BASE_NO 1,IPO_FRAME #BASE,POINT2[] " ",TQ_STATE FALSE}
DECL E6POS XXLX227={X 3178.82104,Y -1687.01099,Z -124.4701,A -38.8299904,B 13.9388504,C -8.95322132,S 2,T 10,E1 -4153.19482,E2 0.0,E3 0.0,E4 0.0,E5 0.0,E6 0.0}
DECL FDAT FXlx227={TOOL_NO 2,BASE_NO 1,IPO_FRAME #BASE,POINT2[] " ",TQ_STATE FALSE}
DECL E6POS XXLX226={X 2377.62109,Y -600.91333,Z -122.117203,A -174.316498,B -60.562809,C -1.327986,S 2,T 42,E1 -4433.27295,E2 0.0,E3 0.0,E4 0.0,E5 0.0,E6 0.0}
DECL FDAT FXlx226={TOOL_NO 2,BASE_NO 1,IPO_FRAME #BASE,POINT2[] " ",TQ_STATE FALSE}
DECL E6POS XXLX225={X 2106.66602,Y -251.165894,Z 213.202896,A 110.725197,B -85.6747131,C 65.7768402,S 2,T 42,E1 -4474.38721,E2 0.0,E3 0.0,E4 0.0,E5 0.0,E6 0.0}
DECL FDAT FXlx225={TOOL_NO 2,BASE_NO 1,IPO_FRAME #BASE,POINT2[] " ",TQ_STATE FALSE}
DECL E6POS XXLX578={X 2064.31494,Y -217.566193,Z 327.9534,A 110.3564,B -85.6859436,C 69.4285126,S 2,T 42,E1 -4474.38477,E2 0.0,E3 0.0,E4 0.0,E5 0.0,E6 0.0}
DECL FDAT FXlx578={TOOL_NO 2,BASE_NO 1,IPO_FRAME #BASE,POINT2[] " ",TQ_STATE FALSE}
DECL PDAT PPDAT1={VEL 100.0,ACC 100.0,APO_DIST 100.0,APO_MODE #CDIS}
DECL SPOT_SUGG_T LAST_SPOT={GUN[] "1                       ",RETR_CMD[] "#CLO                    ",CHOISE[] "#FIRST                  ",CLO_TM[] "1                       ",PGNO1[] "1                       ",PRESS1[] "0                       ",PGNO2[] "1                       ",PRESS2[] "0                       ",SPOT_PARAMS[] "SDAT2                   "}
DECL PDAT PPDAT6={VEL 100.0,ACC 100.0,APO_DIST 100.0,APO_MODE #CDIS}
DECL E6POS XXlx583={X 2066.59204,Y -227.074203,Z 312.509888,A 110.329597,B -85.6865234,C 69.451683,S 2,T 42,E1 -4474.3501,E2 0.0,E3 0.0,E4 0.0,E5 0.0,E6 0.0}
DECL FDAT FXlx583={TOOL_NO 2,BASE_NO 1,IPO_FRAME #BASE,POINT2[] " ",TQ_STATE FALSE}
DECL PDAT PPDAT7={VEL 100.0,ACC 100.0,APO_DIST 100.0,APO_MODE #CDIS}
DECL E6POS XXlx584={X 2065.66895,Y -352.876007,Z 311.141113,A -49.0923691,B -87.7035065,C -128.813095,S 2,T 42,E1 -4219.60986,E2 0.0,E3 0.0,E4 0.0,E5 0.0,E6 0.0}
DECL FDAT FXlx584={TOOL_NO 2,BASE_NO 1,IPO_FRAME #BASE,POINT2[] " ",TQ_STATE FALSE}
DECL E6POS XXLX585={X 2066.68701,Y -527.508118,Z 39.8265114,A -85.7742233,B -55.6886292,C -92.5554199,S 2,T 10,E1 -4219.93799,E2 0.0,E3 0.0,E4 0.0,E5 0.0,E6 0.0}
DECL FDAT FXlx585={TOOL_NO 2,BASE_NO 1,IPO_FRAME #BASE,POINT2[] " ",TQ_STATE FALSE}
DECL PDAT PPDAT8={VEL 100.0,ACC 100.0,APO_DIST 100.0,APO_MODE #CDIS}
DECL E6POS XXLX586={X 2067.14795,Y -570.132324,Z 5.31728601,A -85.6833115,B -56.6240005,C -92.6306229,S 2,T 10,E1 -4219.94092,E2 0.0,E3 0.0,E4 0.0,E5 0.0,E6 0.0}
DECL FDAT FXlx586={TOOL_NO 2,BASE_NO 1,IPO_FRAME #BASE,POINT2[] " ",TQ_STATE FALSE}
DECL PDAT PPDAT9={VEL 100.0,ACC 100.0,APO_DIST 100.0,APO_MODE #CDIS}
DECL E6POS XXLX587={X 2062.77295,Y -616.421997,Z -45.08881,A -86.9156876,B -33.8487091,C -91.7401505,S 2,T 10,E1 -4219.9458,E2 0.0,E3 0.0,E4 0.0,E5 0.0,E6 0.0}
DECL FDAT FXlx587={TOOL_NO 2,BASE_NO 1,IPO_FRAME #BASE,POINT2[] " ",TQ_STATE FALSE}
DECL PDAT PPDAT10={VEL 100.0,ACC 100.0,APO_DIST 100.0,APO_MODE #CDIS}
DECL E6POS XXLX229={X 2207.02002,Y -823.826721,Z -91.6131668,A 90.0196915,B -38.5230598,C 89.9780731,S 2,T 42,E1 -4487.2959,E2 0.0,E3 0.0,E4 0.0,E5 0.0,E6 0.0}
DECL FDAT FXlx229={TOOL_NO 2,BASE_NO 1,IPO_FRAME #BASE,POINT2[] " ",TQ_STATE FALSE}
DECL E6POS XXLX230={X 2063.46704,Y -835.818115,Z -83.1722336,A -87.9995117,B -12.4220896,C -91.1167526,S 2,T 10,E1 -4262.5918,E2 0.0,E3 0.0,E4 0.0,E5 0.0,E6 0.0}
DECL FDAT FXlx230={TOOL_NO 2,BASE_NO 1,IPO_FRAME #BASE,POINT2[] " ",TQ_STATE FALSE}
DECL E6POS XXLX228={X 2056.11108,Y -847.075012,Z -88.9304276,A 89.9993973,B -31.8704395,C 90.0028229,S 2,T 42,E1 -4487.30322,E2 0.0,E3 0.0,E4 0.0,E5 0.0,E6 0.0}
DECL FDAT FXlx228={TOOL_NO 2,BASE_NO 1,IPO_FRAME #BASE,POINT2[] " ",TQ_STATE FALSE}
DECL SPOT_TYPE SS_OLP13={GUN 1,PAIR #FIRST,RETR #CLO,CLO_TM 0,PGNO1 1,PRESS1 1.0,PGNO2 0,PRESS2 0.0}
DECL PDAT PP_OLP41={VEL 100.0,ACC 100.0,APO_DIST 0.0}
DECL SPOT_TYPE SS_OLP14={GUN 1,PAIR #FIRST,RETR #CLO,CLO_TM 0,PGNO1 1,PRESS1 1.0,PGNO2 0,PRESS2 0.0}
DECL E6POS XXLX591={X 2374.73389,Y -849.294922,Z -147.100601,A 90.0008392,B -54.0248108,C 89.9992065,S 2,T 42,E1 -4487.2998,E2 0.0,E3 0.0,E4 0.0,E5 0.0,E6 0.0}
DECL FDAT FXlx591={TOOL_NO 2,BASE_NO 1,IPO_FRAME #BASE,POINT2[] " ",TQ_STATE FALSE}
DECL PDAT PPDAT14={VEL 100.0,ACC 100.0,APO_DIST 100.0,APO_MODE #CDIS}
DECL E6POS XXLX592={X 2065.25806,Y -930.82489,Z -67.1095734,A 90.0008392,B -54.0248108,C 89.9992065,S 2,T 42,E1 -4487.2998,E2 0.0,E3 0.0,E4 0.0,E5 0.0,E6 0.0}
DECL FDAT FXlx592={TOOL_NO 2,BASE_NO 1,IPO_FRAME #BASE,POINT2[] " ",TQ_STATE FALSE}
DECL PDAT PPDAT15={VEL 100.0,ACC 100.0,APO_DIST 100.0,APO_MODE #CDIS}
DECL E6POS XXLX594={X 2622.53906,Y -849.296021,Z -147.097504,A 90.0008316,B -54.0247002,C 89.9993134,S 2,T 42,E1 -4487.2998,E2 0.0,E3 0.0,E4 0.0,E5 0.0,E6 0.0}
DECL FDAT FXlx594={TOOL_NO 2,BASE_NO 1,IPO_FRAME #BASE,POINT2[] " ",TQ_STATE FALSE}
DECL PDAT PPDAT17={VEL 100.0,ACC 100.0,APO_DIST 100.0,APO_MODE #CDIS}
DECL E6POS XXLX595={X 2065.25806,Y -919.828674,Z -49.7837296,A 90.0011292,B -57.6001701,C 89.9989395,S 2,T 42,E1 -4487.2998,E2 0.0,E3 0.0,E4 0.0,E5 0.0,E6 0.0}
DECL FDAT FXlx595={TOOL_NO 2,BASE_NO 1,IPO_FRAME #BASE,POINT2[] " ",TQ_STATE FALSE}
DECL PDAT PPDAT18={VEL 100.0,ACC 100.0,APO_DIST 100.0,APO_MODE #CDIS}
DECL E6POS XXLX596={X 2772.13696,Y -963.370972,Z -700.090515,A -108.568497,B -22.3504105,C -31.4689198,S 2,T 10,E1 -4756.625,E2 0.0,E3 0.0,E4 0.0,E5 0.0,E6 0.0}
DECL FDAT FXlx596={TOOL_NO 2,BASE_NO 1,IPO_FRAME #BASE,POINT2[] " ",TQ_STATE FALSE}
DECL PDAT PPDAT19={VEL 100.0,ACC 100.0,APO_DIST 100.0,APO_MODE #CDIS}
DECL E6POS XXLX609={X 2600.68188,Y -2357.84204,Z 11.5299797,A 15.7114697,B 23.8612595,C 11.6590996,S 2,T 10,E1 -3859.23291,E2 0.0,E3 0.0,E4 0.0,E5 0.0,E6 0.0}
DECL FDAT FXlx609={TOOL_NO 2,BASE_NO 1,IPO_FRAME #BASE,POINT2[] " ",TQ_STATE FALSE}
DECL PDAT PPDAT32={VEL 100.0,ACC 100.0,APO_DIST 100.0,APO_MODE #CDIS}
DECL E6POS XXLX610={X 3228.57397,Y -1264.50903,Z -327.245514,A -61.542881,B 4.42272997,C -3.29499197,S 2,T 10,E1 -3896.23511,E2 0.0,E3 0.0,E4 0.0,E5 0.0,E6 0.0}
DECL FDAT FXlx610={TOOL_NO 2,BASE_NO 1,IPO_FRAME #BASE,POINT2[] " ",TQ_STATE FALSE}
DECL PDAT PPDAT33={VEL 100.0,ACC 100.0,APO_DIST 100.0,APO_MODE #CDIS}
DECL E6POS XXLX611={X 2754.70288,Y -1837.60901,Z 60.1253586,A -39.194561,B 11.7943897,C 5.86210299,S 2,T 2,E1 -3882.32593,E2 0.0,E3 0.0,E4 0.0,E5 0.0,E6 0.0}
DECL FDAT FXlx611={TOOL_NO 2,BASE_NO 1,IPO_FRAME #BASE,POINT2[] " ",TQ_STATE FALSE}
DECL PDAT PPDAT34={VEL 100.0,ACC 100.0,APO_DIST 100.0,APO_MODE #CDIS}
DECL PDAT PP_OLP42={VEL 100.0,ACC 100.0,APO_DIST 0.0}
DECL E6POS XP345={X 2068.52588,Y -424.593414,Z 247.340897,A -84.5327301,B -66.7327805,C -93.6476669,S 2,T 42,E1 -4219.93799,E2 0.0,E3 0.0,E4 0.0,E5 0.0,E6 0.0}
DECL FDAT FP345={TOOL_NO 2,BASE_NO 1,IPO_FRAME #BASE,POINT2[] " ",TQ_STATE FALSE}
DECL PDAT PPDAT37={VEL 100.0,ACC 100.0,APO_DIST 100.0,APO_MODE #CDIS}
DECL E6POS XP346={X 2067.79492,Y -467.097412,Z 187.356598,A -83.7842789,B -70.5107803,C -94.3369293,S 2,T 42,E1 -4219.93799,E2 0.0,E3 0.0,E4 0.0,E5 0.0,E6 0.0}
DECL FDAT FP346={TOOL_NO 2,BASE_NO 1,IPO_FRAME #BASE,POINT2[] " ",TQ_STATE FALSE}
DECL PDAT PPDAT38={VEL 100.0,ACC 100.0,APO_DIST 100.0,APO_MODE #CDIS}
DECL E6POS XP347={X 2117.59204,Y -301.771515,Z 313.628296,A 97.9224091,B -88.4368973,C 82.9338837,S 2,T 42,E1 -4367.44092,E2 0.0,E3 0.0,E4 0.0,E5 0.0,E6 0.0}
DECL FDAT FP347={TOOL_NO 2,BASE_NO 1,IPO_FRAME #BASE,POINT2[] " ",TQ_STATE FALSE}
DECL PDAT PPDAT39={VEL 100.0,ACC 100.0,APO_DIST 100.0,APO_MODE #CDIS}
DECL E6POS XP348={X 2066.9751,Y -1632.005,Z -17.3221703,A 26.6880703,B -15.8931999,C 45.6641693,S 2,T 2,E1 -3882.32788,E2 0.0,E3 0.0,E4 0.0,E5 0.0,E6 0.0}
DECL FDAT FP348={TOOL_NO 2,BASE_NO 1,IPO_FRAME #BASE,POINT2[] " ",TQ_STATE FALSE}
DECL PDAT PPDAT40={VEL 100.0,ACC 100.0,APO_DIST 100.0,APO_MODE #CDIS}
DECL E6POS XP349={X 1967.95203,Y -1296.55603,Z -104.421204,A 20.4034195,B -44.3692703,C 71.2967834,S 2,T 2,E1 -3882.3291,E2 0.0,E3 0.0,E4 0.0,E5 0.0,E6 0.0}
DECL FDAT FP349={TOOL_NO 2,BASE_NO 1,IPO_FRAME #BASE,POINT2[] " ",TQ_STATE FALSE}
DECL PDAT PPDAT41={VEL 100.0,ACC 100.0,APO_DIST 100.0,APO_MODE #CDIS}
DECL E6POS XP350={X 1967.87402,Y -1108.69299,Z -95.3822098,A 7.987391,B -46.6141701,C 82.453743,S 2,T 2,E1 -3882.33008,E2 0.0,E3 0.0,E4 0.0,E5 0.0,E6 0.0}
DECL FDAT FP350={TOOL_NO 2,BASE_NO 1,IPO_FRAME #BASE,POINT2[] " ",TQ_STATE FALSE}
DECL PDAT PPDAT42={VEL 100.0,ACC 100.0,APO_DIST 100.0,APO_MODE #CDIS}
DECL PDAT PPDAT43={VEL 100.0,ACC 100.0,APO_DIST 100.0,APO_MODE #CDIS}
DECL PDAT PPDAT44={VEL 100.0,ACC 100.0,APO_DIST 100.0,APO_MODE #CDIS}
DECL E6POS XP456={X 1967.87,Y -1112.34204,Z -85.6232529,A 7.987535,B -46.61409,C 82.4537582,S 2,T 2,E1 -3882.33105,E2 0.0,E3 0.0,E4 0.0,E5 0.0,E6 0.0}
DECL FDAT FP456={TOOL_NO 2,BASE_NO 1,IPO_FRAME #BASE,POINT2[] " ",TQ_STATE FALSE}
DECL E6POS XP351={X 1904.89905,Y -1156.33899,Z -93.4786224,A 86.2911377,B -74.8139114,C 6.06554317,S 2,T 2,E1 -3882.33203,E2 0.0,E3 0.0,E4 0.0,E5 0.0,E6 0.0}
DECL FDAT FP351={TOOL_NO 2,BASE_NO 1,IPO_FRAME #BASE,POINT2[] " ",TQ_STATE FALSE}
DECL PDAT PPDAT45={VEL 100.0,ACC 100.0,APO_DIST 100.0,APO_MODE #CDIS}
DECL E6POS XP352={X 1899.53003,Y -1126.65295,Z -95.6413498,A 173.313507,B -41.3121986,C -76.1899185,S 2,T 2,E1 -3882.33301,E2 0.0,E3 0.0,E4 0.0,E5 0.0,E6 0.0}
DECL FDAT FP352={TOOL_NO 2,BASE_NO 1,IPO_FRAME #BASE,POINT2[] " ",TQ_STATE FALSE}
DECL PDAT PPDAT46={VEL 100.0,ACC 100.0,APO_DIST 100.0,APO_MODE #CDIS}
DECL PDAT PPDAT47={VEL 100.0,ACC 100.0,APO_DIST 100.0,APO_MODE #CDIS}
DECL E6POS XP455={X 1899.52905,Y -1126.65198,Z -118.918198,A 173.313599,B -41.3121796,C -76.1899414,S 2,T 2,E1 -3882.33301,E2 0.0,E3 0.0,E4 0.0,E5 0.0,E6 0.0}
DECL FDAT FP455={TOOL_NO 2,BASE_NO 1,IPO_FRAME #BASE,POINT2[] " ",TQ_STATE FALSE}
DECL PDAT PPDAT48={VEL 100.0,ACC 100.0,APO_DIST 100.0,APO_MODE #CDIS}
DECL E6POS XP457={X 1903.47498,Y -1325.104,Z -92.6740799,A 150.113098,B -50.6252213,C -42.97715,S 2,T 2,E1 -3880.21704,E2 0.0,E3 0.0,E4 0.0,E5 0.0,E6 0.0}
DECL FDAT FP457={TOOL_NO 2,BASE_NO 1,IPO_FRAME #BASE,POINT2[] " ",TQ_STATE FALSE}
DECL PDAT PPDAT49={VEL 100.0,ACC 100.0,APO_DIST 100.0,APO_MODE #CDIS}
DECL E6POS XP458={X 2066.63599,Y -1759.33801,Z 68.2419968,A 81.0562897,B -24.3322392,C 26.8087902,S 2,T 2,E1 -3880.21704,E2 0.0,E3 0.0,E4 0.0,E5 0.0,E6 0.0}
DECL FDAT FP458={TOOL_NO 2,BASE_NO 1,IPO_FRAME #BASE,POINT2[] " ",TQ_STATE FALSE}
DECL PDAT PPDAT50={VEL 100.0,ACC 100.0,APO_DIST 100.0,APO_MODE #CDIS}
DECL E6POS XSWP_60_5387={X 1790.40796,Y -1122.146,Z -28.0457096,A -179.226395,B -46.9672394,C -90.6360321,S 2,T 2,E1 -3882.33301,E2 0.0,E3 0.0,E4 0.0,E5 0.0,E6 0.0}
DECL FDAT FSWP_60_5387={TOOL_NO 2,BASE_NO 1,IPO_FRAME #BASE,POINT2[] " ",TQ_STATE FALSE}
DECL E6POS XP1={X 2116.1001,Y -2201.521,Z 513.369873,A 72.2993927,B 3.15346503,C 81.6072388,S 6,T 26,E1 -3859.23193,E2 0.0,E3 0.0,E4 0.0,E5 0.0,E6 0.0}
DECL FDAT FP1={TOOL_NO 2,BASE_NO 1,IPO_FRAME #BASE,POINT2[] " ",TQ_STATE FALSE}
DECL PDAT PPDAT53={VEL 100.0,ACC 100.0,APO_DIST 100.0,APO_MODE #CDIS}
DECL PDAT PP_OLP43={VEL 100.0,ACC 100.0,APO_DIST 100.0,APO_MODE #CDIS}
DECL E6POS XXlx231={X 2162.98999,Y -832.758484,Z -85.0697021,A -87.9996033,B -12.4221601,C -91.1167068,S 2,T 10,E1 -4262.5918,E2 0.0,E3 0.0,E4 0.0,E5 0.0,E6 0.0}
DECL FDAT FXlx231={TOOL_NO 2,BASE_NO 1,IPO_FRAME #BASE,POINT2[] " ",TQ_STATE FALSE}
DECL PDAT PP_OLP44={VEL 100.0,ACC 100.0,APO_DIST 100.0,APO_MODE #CDIS}
DECL E6POS XXlx232={X 2207.02002,Y -823.827881,Z -91.6140671,A 90.0197372,B -38.5229683,C 89.9780426,S 2,T 42,E1 -4487.2959,E2 0.0,E3 0.0,E4 0.0,E5 0.0,E6 0.0}
DECL FDAT FXlx232={TOOL_NO 2,BASE_NO 1,IPO_FRAME #BASE,POINT2[] " ",TQ_STATE FALSE}
ENDDAT
